PROGRAM MAIN
VAR
    bdrukknop1 AT %I*: BOOL := FALSE;
    bled1 AT %Q*: BOOL := FALSE;
END_VAR

bled1 := bdrukknop1;

END_PROGRAM

(* stored: Version 1.1.0.1, ProductVersion 3.1.4024.12
   POU MAIN: Id {c6db08f1-aaee-47bf-a939-f814318c1055}, SpecialFunc None *)
